// Mitsubishi GX Developer project: Elevator   PLC: FX1S

PROGRAM MAIN
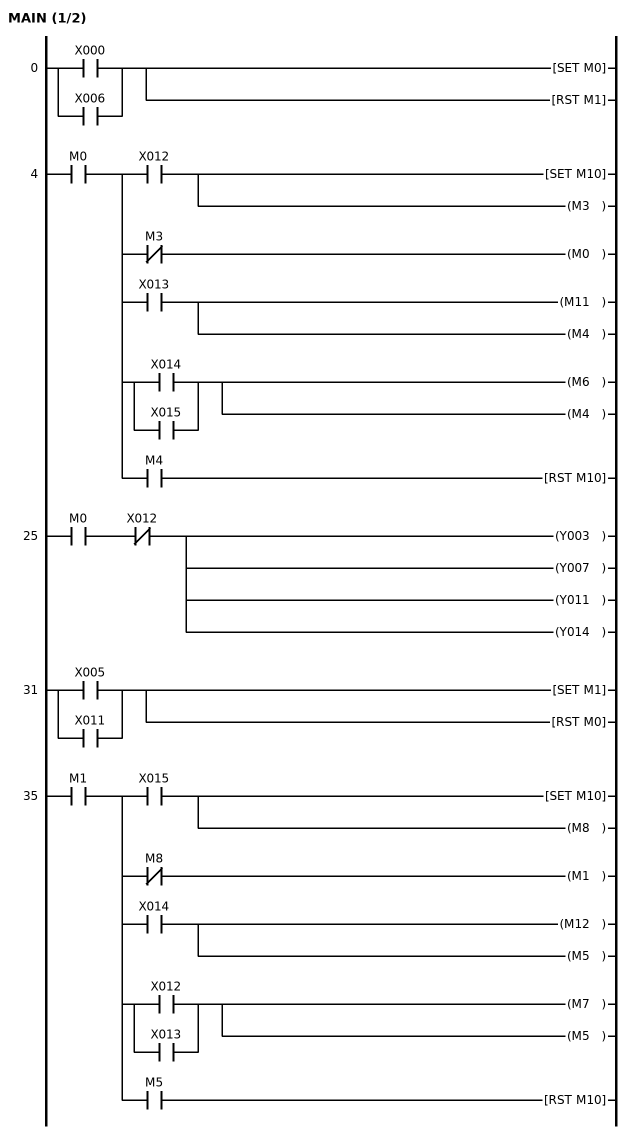
0     LD      X000
      OR      X006
      SET     M0
      RST     M1
4     LD      M0
      MPS
      AND     X012
      SET     M10
      OUT     M3
      MRD
      ANI     M3
      OUT     M0
      MRD
      AND     X013
      OUT     M11
      OUT     M4
      MRD
      LD      X014
      OR      X015
      ANB
      OUT     M6
      OUT     M4
      MPP
      AND     M4
      RST     M10
25    LD      M0
      ANI     X012
      OUT     Y003
      OUT     Y007
      OUT     Y011
      OUT     Y014
31    LD      X005
      OR      X011
      SET     M1
      RST     M0
35    LD      M1
      MPS
      AND     X015
      SET     M10
      OUT     M8
      MRD
      ANI     M8
      OUT     M1
      MRD
      AND     X014
      OUT     M12
      OUT     M5
      MRD
      LD      X012
      OR      X013
      ANB
      OUT     M7
      OUT     M5
      MPP
      AND     M5
      RST     M10
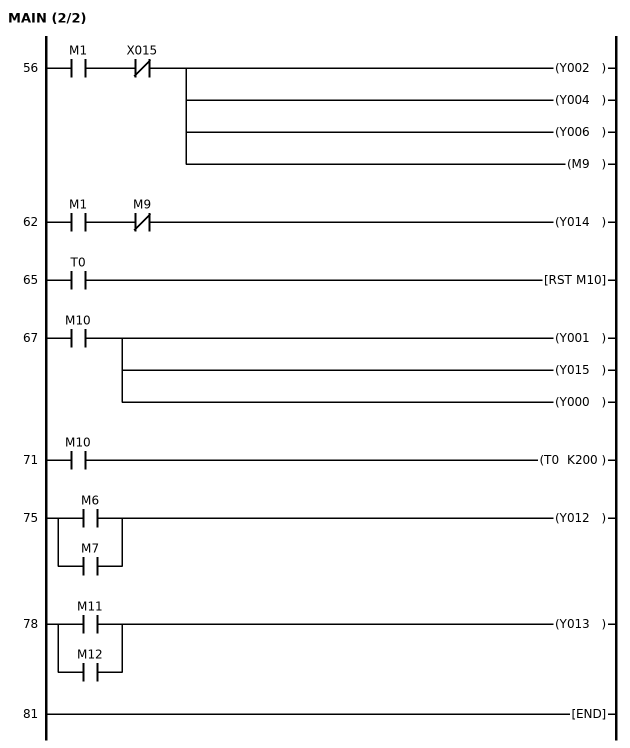
56    LD      M1
      ANI     X015
      OUT     Y002
      OUT     Y004
      OUT     Y006
      OUT     M9
62    LD      M1
      ANI     M9
      OUT     Y014
65    LD      T0
      RST     M10
67    LD      M10
      OUT     Y001
      OUT     Y015
      OUT     Y000
71    LD      M10
      OUT     T0 K200
75    LD      M6
      OR      M7
      OUT     Y012
78    LD      M11
      OR      M12
      OUT     Y013
81    END
END_PROGRAM
